// TwinCAT 3 PLC project Untitled1
// ProgramVersion: 3.1.4023.0
// libraries:
//   Tc2_Standard, * (Beckhoff Automation GmbH)
//   Tc2_System, * (Beckhoff Automation GmbH)
//   Tc2_Utilities, * (Beckhoff Automation GmbH)
//   Tc3_Module, * (Beckhoff Automation GmbH)
//   VisuDialogs, * (System)
//   VisuSymbols,3.5.10.0,System
// project tree:
//   Actuation Systems/Function Blocks/ BulkModulus.TcPOU, DiscreteIntegrator.TcPOU, DiscreteTimeIntegrator_Init.TcPOU, ElectricMotor.TcPOU (not stored), HPU.TcPOU, HydraulicCylinder.TcPOU, OrificeEquation.TcPOU, PressureBuildUp.TcPOU, PressureGradient.TcPOU, Pump.TcPOU (not stored), ValveControlledCylinder.TcPOU, ValveDynamics.TcPOU, VariableBulkModulus.TcPOU
//   Actuation Systems/GVL/ G_ActuationSystems.TcGVL (not stored)
//   Actuation Systems/Programs/ ActuationSystems.TcPOU
//   Functions/ Sign.TcPOU (not stored)
//   / GlobalTextList.TcGTLO, PlcTask.TcTTO, Visualization Manager.TcVMO (not stored)
//   Main Program/ MAIN.TcPOU
//   Parameters/ Param.TcGVL
//   Parameters/Structs/ ST_pValveControlledCylinder.TcDUT
//   VISUs/ Visualization.TcVIS
// real-time tasks:
//   TASK PlcTask: cycle T#100us, priority 20, ADS port 350

CONFIGURATION Untitled1
    RESOURCE PLC ON TwinCAT3
        TASK PlcTask(INTERVAL := T#100us, PRIORITY := 20);
        PROGRAM MAIN WITH PlcTask : MAIN;
    END_RESOURCE
END_CONFIGURATION

// ---- Parameters/Structs/ST_pValveControlledCylinder.TcDUT
TYPE ST_pValveControlledCylinder :
STRUCT
	tCycle : LREAL := 1E-4;
	gravity : LREAL := 9.81;	
	Kv : LREAL := 10 / SQRT(7); 					//[L/min / sqrt(bar)]
	DBore : LREAL := 120E-3;						//[m]
	DRod : LREAL := 80E-3;							//[m]
	xMax : LREAL := 1;								//[m]
	x0 : LREAL := 0.5;								//[m]
	pi : LREAL := 3.14159265359;					//Value of pi
    VA0 : LREAL := 0.01;							//[m^3]
	VB0 : LREAL := 0.01;							//[m^3]
	pMax : LREAL := 200E5; 							//[Pa]
	EffectiveMass : LREAL := 5000;					//[kg]
	ExternalForce : LREAL := EffectiveMass*gravity;	//[N]
	FrictionConstant : LREAL := 10000;				//[N/(m/s)]
	pA0 : LREAL := ExternalForce/0.0113;
	pB0 : LREAL := 1E5;
	pAmax : LREAL :=200E5;
	pBmax : LREAL :=200E5;
	vMax : LREAL := 1; 
	v0 : LREAL := 0; 
	OilBulkModulus : LREAL := 12000E5;					//[Pa]
	AdiatricAirConstant : LREAL := 1.4;				//[-]
	AtmosphericPressure : LREAL := 1.01325E5; 		//[Pa]
	VolumetricAirConstant : LREAL := 0.007;			//[%]
END_STRUCT
END_TYPE

// ---- Parameters/Param.TcGVL
{attribute 'qualified_only'}
VAR_GLOBAL
	pMainJibCylinder : ST_pValveControlledCylinder;
	//pMainKnuckleCylinder : ST_pValveControlledCylinder;
END_VAR

// ---- Main Program/MAIN.TcPOU
PROGRAM MAIN
VAR
	//Integrator
	ssMethodType : SINT := 1; 
	Timer : LREAL;
	
	//Pressure pA
	fbPressureGradient_pA : PressureGradient;
	PressurepA : LREAL;
	
	//Pressure pB
	fbPressureGradient_pB : PressureGradient;
	PressurepB : LREAL;
	
	//Pump
	fbPump : Pump;
	PumpTorque : LREAL;
	PumpFlowRate : LREAL;

	//OrificeEquation QA and QB
	fbOrificeEquationQA : OrificeEquation;
	fbOrificeEquationQB : OrificeEquation;	
	FlowQA : LREAL;
	FlowQB : LREAL;
	
	//HydraulicCylinder
	fbHydraulicCylinder : HydraulicCylinder;
	
	xPos : LREAL;
	ABore : LREAL;
	ARod : LREAL;

(*	pA : LREAL;
	pB : LREAL;
	qA : LREAL;
	qB : LREAL;
	PressureBoreSide : LREAL;
	PressureRodSide : LREAL;
	AreaBoreSide : LREAL;
	AreaRodSide : LREAL;
	LoadForcePistonFL : LREAL;
	FrictionForce : LREAL;		*)
	
	ValveOpeningControl : LREAL := 0.0;
END_VAR

//Timer
Timer := Timer + 0.01;

//Area Cylinder
ABore := EXPT(Param.DBore,2) * (Param.pi/4.0);
ARod := (EXPT(Param.DBore,2) - EXPT(Param.DRod,2)) * (Param.pi/4.0);

//Pump
fbPump(
	MotorSpeedRPM := 413.2,
	PumpDisplacement := 10.6E-6,
	DeltaMaxPressure := 250.0,
	PumpTorque => PumpTorque,
	PumpFlowRate => PumpFlowRate
	);
	
//Pressure Gradient pA and Pressure pA
fbPressureGradient_pA(
	TotalVolume := 0.1E-3 + (fbHydraulicCylinder.PistonPosition * fbHydraulicCylinder.AreaBoreSide),
	BulkModulus := param.BulkModulus,
	FlowrateIn := (FlowQA),
	FlowrateOut := (fbHydraulicCylinder.PistonVelocity * fbHydraulicCylinder.AreaBoreSide),
	PressurePascal => PressurepA		//Pressure
	);
	
//Pressure Gradient pB and Pressure pB
fbPressureGradient_pB(
	TotalVolume := 0.1E-3 + ((param.xMax - fbHydraulicCylinder.PistonPosition) * fbHydraulicCylinder.AreaRodSide),
	BulkModulus := param.BulkModulus,
	FlowrateIn := (fbHydraulicCylinder.PistonVelocity * fbHydraulicCylinder.AreaRodSide),
	FlowrateOut := FlowQB,
	PressurePascal => PressurepB		//Pressure
	);


//OrificeEquationA (Q_A)
fbOrificeEquationQA(
	PressureOut := PressurepA, 			//Found value from old simulink project, this one goes to the tank i guess
	PressureIn := param.pS,	
	Kv := param.Kv,
	ValveOpening := ValveOpeningControl,	
	OrificeFlow => FlowQA
	);
	
//OrificeEquationB (Q_B)
fbOrificeEquationQB(
	PressureOut := param.pT, 			//Found value from old simulink project, this one goes to the tank i guess
	PressureIn := PressurepB,		
	Kv := param.Kv,
	ValveOpening := ValveOpeningControl,
	OrificeFlow => FlowQB
	);
	
//Hydraulic Cylinder 1
fbHydraulicCylinder(
	PistonMass := 5,
	LoadForcePistonFL := 25000*3.14,
	FrictionForce := 10000,
	AreaBoreSide := ABore,
	AreaRodSide := ARod,
	PressureBoreSide := PressurepA,
	PressureRodSide := PressurepB,
	PistonPosition => xPos
	);

END_PROGRAM

// ---- Actuation Systems/Function Blocks/PressureGradient.TcPOU
FUNCTION_BLOCK PressureGradient
VAR_INPUT
	TotalVolume: LREAL;
	BulkModulus: LREAL;
	FlowrateIn: LREAL;
	FlowrateOut: LREAL;
	pMax : LREAL;
	p0 : LREAL;
	param : ST_pValveControlledCylinder;
END_VAR
VAR_OUTPUT
	PressureGradient : LREAL;
	Pressure : LREAL;
END_VAR
VAR
	ssMethodType : SINT := 1; 
	fbPressurePascal : DiscreteTimeIntegrator_Init;
END_VAR

(* Outputs for Atomic SubSystem: '<Root>/PressureGradient' *)
(* Outport: '<Root>/PressureGradientb' incorporates:
 *  Gain: '<S1>/Conv.2'
 *  Product: '<S1>/Product'
 *  Product: '<S1>/Product1'
 *  Sum: '<S1>/Sum' *)
 
//PressureGradient in [Pascal/s]
PressureGradient := (FlowrateIn - FlowrateOut) * (BulkModulus / TotalVolume);
(* End of Outputs for SubSystem: '<Root>/PressureGradient' *)


//Pressure in [Pascal]
fbPressurePascal(
	ssMethodType := ssMethodType,
	tCycle := param.tCycle,
	In := PressureGradient,
	Init := p0,
	minOut := G_ActuationSystems.ReturnPressure,
	maxOut := param.pAmax,
	Out => Pressure
	);

END_FUNCTION_BLOCK

// ---- Actuation Systems/Function Blocks/BulkModulus.TcPOU
FUNCTION_BLOCK BulkModulus
VAR_INPUT
END_VAR
VAR_OUTPUT
	BulkModulus : LREAL := 10000E5;
END_VAR
VAR
END_VAR

END_FUNCTION_BLOCK

// ---- Actuation Systems/Function Blocks/DiscreteTimeIntegrator_Init.TcPOU
FUNCTION_BLOCK DiscreteTimeIntegrator_Init
VAR_INPUT
	ssMethodType: SINT;
	In: LREAL;
	Init: LREAL;
	minOut : LREAL;
	maxOut : LREAL;
	tCycle : LREAL;
END_VAR
VAR_OUTPUT
	Out: LREAL;
END_VAR
VAR
	c_DiscreteTimeIntegrator_IC: USINT;
	c_DiscreteTimeIntegrator_DS: LREAL;
END_VAR



CASE ssMethodType OF
    0: 
        (* SystemInitialize for Atomic SubSystem: '<Root>/DiscreteTimeIntegrator_Init' *)
        (* InitializeConditions for DiscreteIntegrator: '<S1>/Discrete-Time Integrator' *)
        c_DiscreteTimeIntegrator_IC := 1;
        (* End of SystemInitialize for SubSystem: '<Root>/DiscreteTimeIntegrator_Init' *)
    1: 
        (* Outputs for Atomic SubSystem: '<Root>/DiscreteTimeIntegrator_Init' *)
        (* DiscreteIntegrator: '<S1>/Discrete-Time Integrator' *)

        IF c_DiscreteTimeIntegrator_IC <> 0 THEN 
            c_DiscreteTimeIntegrator_DS := Init;

            IF c_DiscreteTimeIntegrator_DS >= maxOut THEN 
                c_DiscreteTimeIntegrator_DS := maxOut;
            ELSIF c_DiscreteTimeIntegrator_DS <= minOut THEN 
                c_DiscreteTimeIntegrator_DS := minOut;
            END_IF;

        END_IF;


        IF c_DiscreteTimeIntegrator_DS >= maxOut THEN 
            c_DiscreteTimeIntegrator_DS := maxOut;
        ELSIF c_DiscreteTimeIntegrator_DS <= minOut THEN 
            c_DiscreteTimeIntegrator_DS := minOut;
        END_IF;

        (* Outport: '<Root>/Out' incorporates:
         *  DiscreteIntegrator: '<S1>/Discrete-Time Integrator' *)
        Out := c_DiscreteTimeIntegrator_DS;
        (* Update for DiscreteIntegrator: '<S1>/Discrete-Time Integrator' *)
        c_DiscreteTimeIntegrator_IC := 0;
        c_DiscreteTimeIntegrator_DS := (tCycle * In) + c_DiscreteTimeIntegrator_DS;

        IF c_DiscreteTimeIntegrator_DS >= maxOut THEN 
            c_DiscreteTimeIntegrator_DS := maxOut;
        ELSIF c_DiscreteTimeIntegrator_DS <= minOut THEN 
            c_DiscreteTimeIntegrator_DS := minOut;
        END_IF;

        (* End of Update for DiscreteIntegrator: '<S1>/Discrete-Time Integrator' *)
        (* End of Outputs for SubSystem: '<Root>/DiscreteTimeIntegrator_Init' *)
END_CASE;

END_FUNCTION_BLOCK

// ---- Actuation Systems/Function Blocks/OrificeEquation.TcPOU
FUNCTION_BLOCK OrificeEquation
VAR_INPUT
	PressureOut: LREAL;
	PressureIn: LREAL;
	ValveOpening: LREAL;
	param : ST_pValveControlledCylinder;
END_VAR
VAR_OUTPUT
	OrificeFlow: LREAL;
END_VAR
VAR
	rtb_Sum: LREAL;
	y: LREAL;
	temp1: LREAL;

END_VAR


(* Outputs for Atomic SubSystem: '<Root>/OrificeEquation' *)
(* Sum: '<S1>/Sum' *)
rtb_Sum := (PressureIn - PressureOut)*1E-5;
(* Signum: '<S1>/Sign' *)

IF rtb_Sum < 0.0 THEN 
    y := -1.0;
ELSIF rtb_Sum > 0.0 THEN 
    y := 1.0;
ELSE 
    y := rtb_Sum;
END_IF;

(* End of Signum: '<S1>/Sign' *)

(* Outport: '<Root>/OrificeFlow' incorporates:
 *  Abs: '<S1>/Abs'
 *  Product: '<S1>/Product2'
 *  Sqrt: '<S1>/Sqrt1' *)
temp1 := ABS(rtb_Sum);
OrificeFlow := (((param.Kv * ValveOpening) * y) * SQRT(temp1)) * (1/60000);
(* End of Outputs for SubSystem: '<Root>/OrificeEquation' *)

END_FUNCTION_BLOCK

// ---- Actuation Systems/Function Blocks/HydraulicCylinder.TcPOU
FUNCTION_BLOCK HydraulicCylinder
VAR_INPUT
	PressureBoreSide: LREAL;
	PressureRodSide: LREAL;
	Aa: LREAL;
	Ab: LREAL;
	param : ST_pValveControlledCylinder;
END_VAR
VAR_OUTPUT
	PistonAcceleration: LREAL;
	PistonVelocity : LREAL;
	PistonPosition : LREAL;
END_VAR
VAR
	ssMethodType : SINT := 1; 
	fbPistonVelocity : DiscreteTimeIntegrator_Init;
	fbPistonPosition : DiscreteTimeIntegrator_Init;

END_VAR


(* Outputs for Atomic SubSystem: '<Root>/HydraulicCylinder' *)
(* Outport: '<Root>/PistonAcceleration' incorporates:
 *  Gain: '<S1>/Gain1'
 *  Gain: '<S1>/Gain2'
 *  Product: '<S1>/Divide '
 *  Product: '<S1>/Product'
 *  Product: '<S1>/Product1'
 *  Sum: '<S1>/sum' *)
 
//Area Cylinder
Aa := EXPT(param.DBore,2) * (param.pi/4.0);
Ab := (EXPT(param.DBore,2) - EXPT(param.DRod,2)) * (param.pi/4.0);
 
PistonAcceleration := ((PressureBoreSide * Aa) - (PressureRodSide * Ab) - param.FrictionConstant*PistonVelocity - param.ExternalForce) / param.EffectiveMass;
(* End of Outputs for SubSystem: '<Root>/HydraulicCylinder' *)

fbPistonVelocity(
	ssMethodType := ssMethodType,
	In := PistonAcceleration,
	Init := param.v0,
	minOut := -param.vMax,
	maxOut := param.vMax,
	Out => PistonVelocity
	);
	
fbPistonPosition(
	ssMethodType := ssMethodType,
	In := PistonVelocity,
	Init := param.x0,
	minOut := 0,
	maxOut := param.xMax,
	Out => PistonPosition
	);

IF PistonPosition >= param.xMax THEN 
	PistonPosition := param.xMax;
ELSIF PistonPosition <= 0 THEN 
	PistonPosition := 0;
END_IF;

END_FUNCTION_BLOCK

// ---- Actuation Systems/Function Blocks/DiscreteIntegrator.TcPOU
FUNCTION_BLOCK DiscreteIntegrator
VAR_INPUT
	ssMethodType: SINT;
	In1: LREAL;
	StepTime : LREAL := 0.001;
END_VAR
VAR_OUTPUT
	Out1: LREAL;
END_VAR
VAR
	c_DiscreteIntegratorMain_DS: LREAL;
	k1: LREAL := 1.0;

END_VAR



CASE ssMethodType OF
    0: 
        (* SystemInitialize for Atomic SubSystem: '<Root>/DiscreteIntegrator' *)
        (* InitializeConditions for DiscreteIntegrator: '<S1>/DiscreteIntegratorMain' *)
        c_DiscreteIntegratorMain_DS := 0.0;
        (* End of SystemInitialize for SubSystem: '<Root>/DiscreteIntegrator' *)
    1: 
        (* Outputs for Atomic SubSystem: '<Root>/DiscreteIntegrator' *)
        (* Outport: '<Root>/Out1' incorporates:
         *  DiscreteIntegrator: '<S1>/DiscreteIntegratorMain' *)
        Out1 := c_DiscreteIntegratorMain_DS;
        (* Update for DiscreteIntegrator: '<S1>/DiscreteIntegratorMain' incorporates:
         *  Gain: '<S1>/Gain' *)
        c_DiscreteIntegratorMain_DS := ((k1 * In1) * StepTime) + c_DiscreteIntegratorMain_DS;
        (* End of Outputs for SubSystem: '<Root>/DiscreteIntegrator' *)
		

END_CASE;

END_FUNCTION_BLOCK

// ---- Actuation Systems/Function Blocks/HPU.TcPOU
FUNCTION_BLOCK HPU
VAR_INPUT
	par : ST_pValveControlledCylinder;
END_VAR
VAR_OUTPUT
	TankPressure : LREAL;
	SupplyPressure : LREAL;
END_VAR
VAR
	//Pump
	fbPump : Pump;
	PumpTorque : LREAL;
	PumpFlowRate : LREAL;
END_VAR


//Pump
fbPump(
MotorSpeedRPM := 413.2,
PumpDisplacement := 10.6E-6,
DeltaMaxPressure := 250.0,
PumpTorque => PumpTorque,
PumpFlowRate => PumpFlowRate
);

TankPressure := 1.2E5;
SupplyPressure := 180E5; 

G_ActuationSystems.ReturnPressure := TankPressure;
G_ActuationSystems.SupplyPressure := SupplyPressure;

END_FUNCTION_BLOCK

// ---- Actuation Systems/Function Blocks/PressureBuildUp.TcPOU
FUNCTION_BLOCK PressureBuildUp
VAR
	fbPressureGradient : PressureGradient;
	fbDiscreteIntegrator : DiscreteIntegrator;
	
	IntegratorIn : LREAL;
	IntegratorOut : LREAL;
	ssMethodType : SINT := 1; 
	

//	fbPressure : DiscreteIntegrator;
//	fbPressureGradient : PressureGradient;
END_VAR
VAR_INPUT
	TotalVolume1 : LREAL;
	FlowrateIn1 : LREAL;
	FlowrateOut1 : LREAL;
	par : ST_pValveControlledCylinder;
END_VAR
VAR_OUTPUT
//	PressureBar : LREAL;
//	PressurePascal : LREAL;
END_VAR


fbPressureGradient(
	TotalVolume := TotalVolume1,
	FlowrateIn := FlowrateIn1,
	FlowrateOut := FlowrateOut1
	);

//pA
(* fbPressure(
	ssMethodType := ssMethodType,
	In1 := fbPressureGradient.PressureGradientPascal,
	Out1 => PressurePascal
	);
	
PressureGradientPascal := PressureGradientBar*1E5;      //Multiplies to get Pascal *)

END_FUNCTION_BLOCK

// ---- Actuation Systems/Function Blocks/ValveControlledCylinder.TcPOU
FUNCTION_BLOCK ValveControlledCylinder
VAR_INPUT
	ReturnPressure : LREAL;
	SupplyPressure : LREAL;
	par : ST_pValveControlledCylinder;
END_VAR
VAR_OUTPUT
	PistonArea : LREAL;
	AnnulusArea : LREAL;
END_VAR
VAR

//Pressure pA
fbPressureGradient_pA : PressureGradient;
PressurepA : LREAL;

//Pressure pB
fbPressureGradient_pB : PressureGradient;
PressurepB : LREAL;

//OrificeEquation QA and QB
fbOrificeEquationQ_P_A : OrificeEquation;
fbOrificeEquationQ_B_R : OrificeEquation;
fbOrificeEquationQ_P_B : OrificeEquation;
fbOrificeEquationQ_A_R : OrificeEquation;	
FlowQ_P_A : LREAL;
FlowQ_B_R : LREAL;	
FlowQ_P_B : LREAL;
FlowQ_A_R : LREAL;
FlowQA : LREAL;
FlowQB : LREAL;
FlowQL : LREAL := 0.00001;

//HydraulicCylinder
fbHydraulicCylinder : HydraulicCylinder;

xPos : LREAL;
ValveOpeningControl : LREAL := 0.0;
uDcv : LREAL := 0.0;
uDcvEnable : BOOL := TRUE; 

fbBulkModulus : BulkModulus;
fbVariableBulkModulus : VariableBulkModulus;

END_VAR


IF uDcvEnable THEN
	ValveOpeningControl := uDcv;
ELSE 
	ValveOpeningControl := 0;
END_IF

//VariableBulkModulus
fbVariableBulkModulus(
	OilBulkModulus := par.OilBulkModulus,
	AdiatricAirConstant := par.AdiatricAirConstant,
	AtmosphericPressure := par.AtmosphericPressure,
	VolumetricAirContentOfOil := par.VolumetricAirConstant
	);

//Pressure Gradient pA and Pressure pA
fbPressureGradient_pA(
	TotalVolume := par.VA0 + (fbHydraulicCylinder.PistonPosition * fbHydraulicCylinder.Aa),
	BulkModulus := fbBulkModulus.BulkModulus,
	FlowrateIn := FlowQA,
	FlowrateOut := (fbHydraulicCylinder.PistonVelocity * fbHydraulicCylinder.Aa),
	p0 := par.pA0,
	param := par,
	Pressure => PressurepA		
	);

//Pressure Gradient pB and Pressure pB
fbPressureGradient_pB(
	TotalVolume := par.VB0 + ((par.xMax - fbHydraulicCylinder.PistonPosition) * fbHydraulicCylinder.Ab),
	BulkModulus := fbBulkModulus.BulkModulus,
	FlowrateIn := (fbHydraulicCylinder.PistonVelocity * fbHydraulicCylinder.Ab),
	FlowrateOut := FlowQB + FlowQL,
	p0 := par.pB0,
	param := par,
	Pressure => PressurepB		
	);

//Flow through orifices Q_P_A, Q_A_R, Q_B_R, Q_P_B
fbOrificeEquationQ_P_A(
	PressureOut := PressurepA, 			
	PressureIn := SupplyPressure,	
	ValveOpening := ValveOpeningControl,	
	param := par,
	OrificeFlow => FlowQ_P_A
	);
	
fbOrificeEquationQ_A_R(
	PressureOut := ReturnPressure, 			
	PressureIn :=  PressurepA,	
	ValveOpening := ValveOpeningControl,	
	param := par,
	OrificeFlow => FlowQ_A_R
	);

fbOrificeEquationQ_B_R(
	PressureOut := ReturnPressure, 			
	PressureIn := PressurepB,			
	ValveOpening := ValveOpeningControl,
	param := par,
	OrificeFlow => FlowQ_B_R
	);
	
fbOrificeEquationQ_P_B(
	PressureOut := PressurepB, 			
	PressureIn := SupplyPressure,			
	ValveOpening := ValveOpeningControl,
	param := par,
	OrificeFlow => FlowQ_P_B
	);	

IF ValveOpeningControl > 0 THEN
	FlowQA := FlowQ_P_A;		
	FlowQB := FlowQ_B_R;
ELSIF ValveOpeningControl < 0 THEN
	FlowQA := FlowQ_A_R;		
	FlowQB := FlowQ_P_B;
ELSE
	FlowQA := 0.0;		
	FlowQB := 0.0;	
END_IF

	
//Hydraulic Cylinder 1
fbHydraulicCylinder(
	PressureBoreSide := PressurepA,
	PressureRodSide := PressurepB,
	Aa => PistonArea,
	Ab => AnnulusArea,
	PistonPosition => xPos,
	param := Param.pMainJibCylinder
	);

END_FUNCTION_BLOCK

// ---- Actuation Systems/Function Blocks/VariableBulkModulus.TcPOU
FUNCTION_BLOCK VariableBulkModulus
VAR_INPUT
	OilBulkModulus: LREAL;
	AdiatricAirConstant: LREAL;
	AtmosphericPressure: LREAL;
	CapacitancePressure: LREAL;
	VolumetricAirContentOfOil: LREAL;
END_VAR
VAR_OUTPUT
	VariableBulkModulus: LREAL;
END_VAR
VAR
	rtb_Add: LREAL;
END_VAR

rtb_Add := AtmosphericPressure + CapacitancePressure;

VariableBulkModulus := 1.0 / ((1.0 / OilBulkModulus) - (1.0 / ((((VolumetricAirContentOfOil - 1.0) / (EXPT(AtmosphericPressure / rtb_Add, 1.0 / AdiatricAirConstant) * VolumetricAirContentOfOil)) - 1.0) * (rtb_Add * AdiatricAirConstant))));

END_FUNCTION_BLOCK

// ---- Actuation Systems/Function Blocks/ValveDynamics.TcPOU
FUNCTION_BLOCK ValveDynamics
VAR_INPUT
END_VAR
VAR_OUTPUT
END_VAR
VAR
END_VAR

END_FUNCTION_BLOCK

// ---- Actuation Systems/Programs/ActuationSystems.TcPOU
PROGRAM ActuationSystems
VAR
fbMainJibCylinder : ValveControlledCylinder;
//fbKnuckleJibCylinder : ValveControlledCylinder;
fbHPU : HPU;
END_VAR


fbHPU(
);

fbMainJibCylinder(
ReturnPressure := G_ActuationSystems.ReturnPressure,
SupplyPressure := G_ActuationSystems.SupplyPressure,
par := Param.pMainJibCylinder
);

(* fbKnuckleJibCylinder(
ReturnPressure := G_ActuationSystems.ReturnPressure,
SupplyPressure := G_ActuationSystems.SupplyPressure,
par := Param.pMainKnuckleCylinder
); *)

END_PROGRAM

// ---- GlobalTextList.TcGTLO
TEXTLIST GlobalTextList
  398 = '%0.1f'
  566 = '%0.2f'
  627 = '%0.5f'
  729 = '%2f'
  210 = '%f'
  839 = '%f.2'
  735 = '%f0.2'
  760 = '%f0.5'
  189 = '%f2'
  842 = '0'
  716 = 'x = 0'
END_TEXTLIST

// ---- VISUs/Visualization.TcVIS
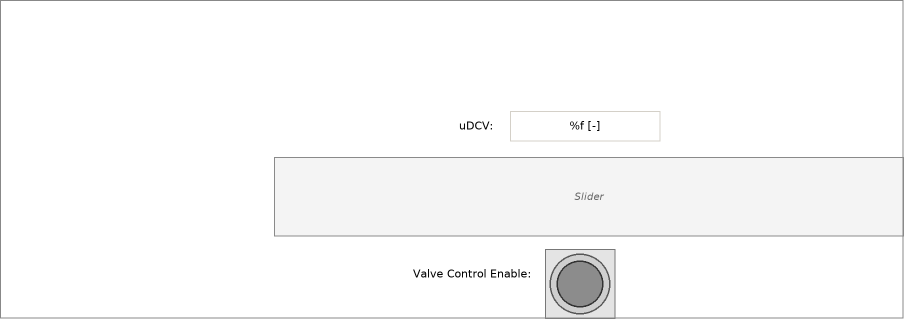
VISUALIZATION Visualization  // 904x319
    Slider (274,157 630x79), variable: ActuationSystems.fbMainJibCylinder.uDcv, scale -1..1
    PushSwitchLed (545,249 70x70), variable: ActuationSystems.fbMainJibCylinder.uDcvEnable, behaviour: TOGGLE, style: Switch-PushSwitchLed-Gray
    Textfield (510,111 150x30), "%f [-]", text variable: ActuationSystems.fbMainJibCylinder.uDcv
        OnMouseClick: write the text variable via Default, min -1, max 1
    Label (443,111 66x30), "uDCV:"
    Label (381,259 182x30), "Valve Control Enable:"
END_VISUALIZATION
